// TIA Portal V16 export
// export: Created 2022-11-17T15:49:42.114243Z, ExportSetting WithDefaults, DisplayName Totally Integrated Automation Portal, DisplayVersion V16 Update 6, DisplayName TIA Portal Version Control Interface, DisplayVersion V16 Update 2, DisplayName TIA Portal Openness, DisplayVersion V16 Update 6, DisplayName SINAMICS Startdrive Advanced, DisplayVersion V16 Update 5, DisplayName SINAMICS Startdrive G130, G150, S120, S150, SINAMICS MV, S210, DisplayVersion V16 Update 5, DisplayName SINAMICS Startdrive G110M, G120, G120C, G120D, G120P, G115D, DisplayVersion V16 Update 5, DisplayName STEP 7 Professional, DisplayVersion V16 Update 6, DisplayName STEP 7 Safety, DisplayVersion V16, DisplayName WinCC Advanced, DisplayVersion V16 Update 6
DATA_BLOCK "Inverter_Data"   // DB210
{ S7_Optimized_Access := 'FALSE' }
VERSION : 0.1
// stored: AutoNumber false, IsOnlyStoredInLoadMemory false, IsWriteProtectedInAS false
   VAR
      U201 { S7_SetPoint := 'True'} : "InverterData";
      U221 { S7_SetPoint := 'True'} : "InverterData";
      U241 { S7_SetPoint := 'True'} : "InverterData";
      U261 { S7_SetPoint := 'True'} : "InverterData";
      U321 { S7_SetPoint := 'True'} : "InverterData";
   END_VAR
BEGIN
   U201.control_word := 16#047A;
   U201.setpoint := 0.0;
   U201.ref_quantity.speed_p2000 := 3000.0;
   U201.ref_quantity.current_p2002 := 5.0;
   U201.ref_quantity.torque_p2003 := 7.61;
   U201.status_word := 16#EB40;
   U201.actual_speed := 0.0;
   U201.actual_current := 0.0;
   U201.actual_torque := 0.0;
   U201.actual_alarm := 16#0000;
   U201.actual_fault := 16#0000;
   U201.RETVAL_RD := 16#0000;
   U201.RETVAL_WR := 16#0000;
   U221.control_word := 16#047E;
   U221.setpoint := 0.0;
   U221.ref_quantity.speed_p2000 := 3000.0;
   U221.ref_quantity.current_p2002 := 1.86;
   U221.ref_quantity.torque_p2003 := 3.59;
   U221.status_word := 16#EB31;
   U221.actual_speed := 0.0;
   U221.actual_current := 0.001702881;
   U221.actual_torque := 0.0;
   U221.actual_alarm := 16#0000;
   U221.actual_fault := 16#0000;
   U221.RETVAL_RD := 16#0000;
   U221.RETVAL_WR := 16#0000;
   U241.control_word := 16#047E;
   U241.setpoint := 0.0;
   U241.ref_quantity.speed_p2000 := 3000.0;
   U241.ref_quantity.current_p2002 := 1.86;
   U241.ref_quantity.torque_p2003 := 3.59;
   U241.status_word := 16#EB31;
   U241.actual_speed := 0.0;
   U241.actual_current := 0.002043457;
   U241.actual_torque := 0.0;
   U241.actual_alarm := 16#0000;
   U241.actual_fault := 16#0000;
   U241.RETVAL_RD := 16#0000;
   U241.RETVAL_WR := 16#0000;
   U261.control_word := 16#047E;
   U261.setpoint := 0.0;
   U261.ref_quantity.speed_p2000 := 3000.0;
   U261.ref_quantity.current_p2002 := 1.86;
   U261.ref_quantity.torque_p2003 := 3.59;
   U261.status_word := 16#EB31;
   U261.actual_speed := 0.0;
   U261.actual_current := 0.0;
   U261.actual_torque := 0.0;
   U261.actual_alarm := 16#0000;
   U261.actual_fault := 16#0000;
   U261.RETVAL_RD := 16#0000;
   U261.RETVAL_WR := 16#0000;
   U321.control_word := 16#047E;
   U321.setpoint := 0.0;
   U321.ref_quantity.speed_p2000 := 3000.0;
   U321.ref_quantity.current_p2002 := 6.9;
   U321.ref_quantity.torque_p2003 := 29.5;
   U321.status_word := 16#EB31;
   U321.actual_speed := 0.0;
   U321.actual_current := 0.0;
   U321.actual_torque := 0.0;
   U321.actual_alarm := 16#0000;
   U321.actual_fault := 16#0000;
   U321.RETVAL_RD := 16#0000;
   U321.RETVAL_WR := 16#0000;
END_DATA_BLOCK
